FUNCTION_BLOCK RunLoading EXTENDS RunUnitSlave
VAR_INPUT
	externalSlotValid  : BOOL;
	isSlotValidOverride : BOOL; //eniginnering use , dry run
END_VAR
VAR_OUTPUT
	purgeRequest AT%Q* : BOOL; //link to SCARA2
END_VAR
VAR	
	existence : POINTER TO RunSignal;	
	watchDog : TON;
END_VAR
VAR PERSISTENT
	currentId : DWORD;
END_VAR

SUPER^();

//signal reset
IF previousNode<>0 AND_THEN NOT previousNode^.isPurged THEN
		purgeRequest :=FALSE;
END_IF

//-------------------------------
//	Slot-1 to loading bottom part
//-------------------------------

CASE outputState OF
	eSpecialStates.INITIAL_BEGIN:
		NextState := eSpecialStates.INITIAL_END;
	//---------------------
	//	Working
	//---------------------
	eSpecialStates.SLAVE_ENTER_PROCEDURE:
		//check if empty
		bSerialTransition := existence^.debouncedOff;
		IF bSerialTransition THEN
			
			IF previousNode<>0 AND_THEN previousNode^.isPurged THEN
				purgeRequest :=TRUE;
			END_IF
			SlotBase^.Valid := FALSE; //always false in beginning
			slaveWorkingSignal[1] := TRUE; // trigger scara to put
		END_IF
	16#201:
		bSerialTransition := NOT slaveWorkingSignal[1]; //scara should set valid before reset working 
		IF bSerialTransition THEN
			SlotBase^.Valid := externalSlotValid OR isSlotValidOverride; //transit
		END_IF
	16#202:
		//check if material status matched sensor status
		bSerialTransition := (SlotBase^.Valid = existence^.debouncedOn) OR isSlotValidOverride;
		IF bSerialTransition AND purgeRequest AND NOT SlotBase^.Valid THEN
			//SCARA2 had received purge request and no longer loading the parts
			isPurged := TRUE;
			watchDog.IN := FALSE;
			
			//give material id
			SlotBase^.Id := currentId;
			currentId := currentId+1;
			IF currentId >= DWORD#16#FFFFFFFF THEN
				currentId := 0;
			END_IF
			
		ELSIF watchDog.Q THEN
			//TODO ,raise alarm
		END_IF
		watchDog.IN := TRUE; //activate
	16#203:
		NextState := eSpecialStates.SLAVE_WORK_DONE;
END_CASE

METHOD FB_init : BOOL
VAR_INPUT
	bInitRetains : BOOL; // if TRUE, the retain variables are initialized (warm start / cold start)
	bInCopyCode : BOOL;  // if TRUE, the instance afterwards gets moved into the copy code (online change)
	
	argParent : POINTER TO RunUnitGeneric;
	argSlotBase : POINTER TO RunMaterial;
	argSlotLast : POINTER TO RunMaterial;
	
	argWorkingSignal : POINTER TO BOOL;
	
	argExistence : POINTER TO RunSignal;
END_VAR
//initialize 
Parent := argParent;
SlotBase := argSlotBase;
SlotLast := argSlotLast;
//
IF bInitRetains THEN
	NextState := eSpecialStates.INITIAL_BEGIN;
END_IF

workingSignal := argWorkingSignal; //link

existence := argExistence;
END_METHOD

END_FUNCTION_BLOCK

(* stored: Version 1.1.0.1, ProductVersion 3.1.4024.0
   POU RunLoading: Id {0885f03e-fd54-45c2-8cc3-34c2d157a6e9}, SpecialFunc None
   Method FB_init: Id {73f2038d-f762-4ac2-a699-acb024b4c517} *)
